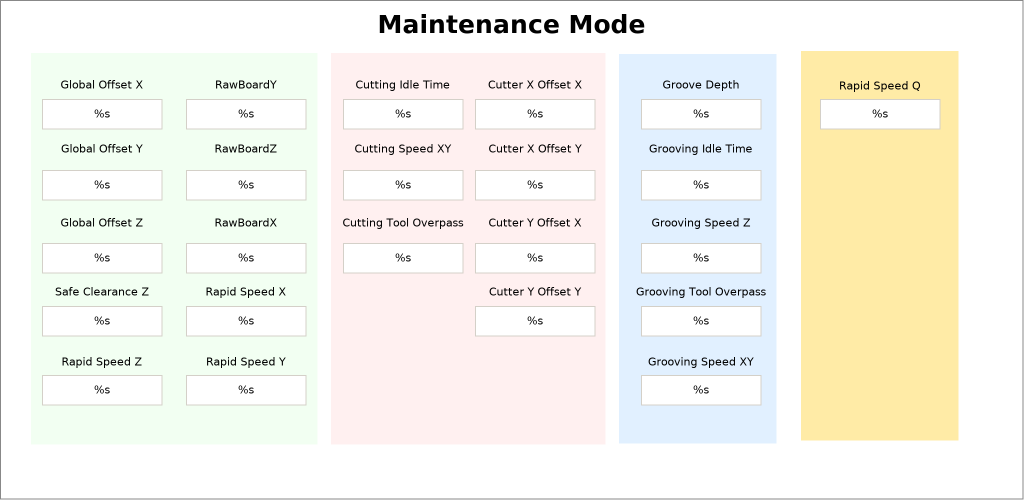
VISUALIZATION V_MaintenanceMode  // 1024x500
VAR_IN_OUT
	HMI : ST_PackMLBaseModule_HMI;
	HMI_GantryXYZ : ST_GantryXYZ_HMI;
	HMI_Recipe : ST_RecipeBuilder_HMI;
END_VAR
    Rectangle (30,52 288x393)
    Rectangle (330,52 276x393)
    Label (0,-1 1023x50), "Maintenance Mode"
    Rectangle (618,53 159x391)
    Textfield (641,99 120x30), "%s", text variable: HMI_Recipe.Config.GrooveDepthZ
        OnMouseClick: write the text variable via VisuDialogs.Numpad, min HMI_Recipe.Limits.GrooveDepthZ.MinVal, max HMI_Recipe.Limits.GrooveDepthZ.MaxVal
    Label (641,70 120x30), "Groove Depth"
    Textfield (641,306 120x30), "%s", text variable: HMI_Recipe.Config.GroovingOverpass
        OnMouseClick: write the text variable via VisuDialogs.Numpad, min HMI_Recipe.Limits.GroovingOverpass.MinVal, max HMI_Recipe.Limits.GroovingOverpass.MaxVal
    Label (641,277 120x30), "Grooving Tool Overpass"
    Textfield (641,375 120x30), "%s", text variable: HMI_GantryXYZ.Config.GroovingSpeedXY
        OnMouseClick: write the text variable via VisuDialogs.Numpad, min HMI_GantryXYZ.Limits.GroovingSpeedXY.MinVal, max HMI_GantryXYZ.Limits.GroovingSpeedXY.MaxVal
    Label (641,347 120x30), "Grooving Speed XY"
    Textfield (186,306 120x30), "%s", text variable: HMI_GantryXYZ.Config.RapidSpeedX
        OnMouseClick: write the text variable via VisuDialogs.Numpad, min HMI_GantryXYZ.Limits.RapidSpeedX.MinVal, max HMI_GantryXYZ.Limits.RapidSpeedX.MaxVal
    Label (186,277 120x30), "Rapid Speed X"
    Textfield (186,375 120x30), "%s", text variable: HMI_GantryXYZ.Config.RapidSpeedY
        OnMouseClick: write the text variable via VisuDialogs.Numpad, min HMI_GantryXYZ.Limits.RapidSpeedY.MinVal, max HMI_GantryXYZ.Limits.RapidSpeedY.MaxVal
    Label (186,347 120x30), "Rapid Speed Y"
    Textfield (641,243 120x30), "%s", text variable: HMI_GantryXYZ.Config.GroovingSpeedZ
        OnMouseClick: write the text variable via VisuDialogs.Numpad, min HMI_GantryXYZ.Limits.GroovingSpeedZ.MinVal, max HMI_GantryXYZ.Limits.GroovingSpeedZ.MaxVal
    Label (641,208 120x30), "Grooving Speed Z"
    Textfield (42,375 120x30), "%s", text variable: HMI_GantryXYZ.Config.RapidSpeedZ
        OnMouseClick: write the text variable via VisuDialogs.Numpad, min HMI_GantryXYZ.Limits.RapidSpeedZ.MinVal, max HMI_GantryXYZ.Limits.RapidSpeedZ.MaxVal
    Label (42,347 120x30), "Rapid Speed Z"
    Textfield (641,170 120x30), "%s", text variable: HMI_GantryXYZ.Config.GroovingIdleTime
        OnMouseClick: write the text variable via VisuDialogs.Numpad, min HMI_GantryXYZ.Limits.GroovingIdleTime.MinVal, max HMI_GantryXYZ.Limits.GroovingIdleTime.MaxVal
    Label (641,134 120x30), "Grooving Idle Time"
    Label (343,134 120x30), "Cutting Speed XY"
    Textfield (343,243 120x30), "%s", text variable: HMI_Recipe.Config.CuttingOverpass
        OnMouseClick: write the text variable via VisuDialogs.Numpad, min HMI_Recipe.Limits.CuttingOverpass.MinVal, max HMI_Recipe.Limits.CuttingOverpass.MaxVal
    Label (343,208 120x30), "Cutting Tool Overpass"
    Textfield (343,99 120x30), "%s", text variable: HMI_GantryXYZ.Config.CuttingIdleTime
        OnMouseClick: write the text variable via VisuDialogs.Numpad, min HMI_GantryXYZ.Limits.CuttingIdleTime.MinVal, max HMI_GantryXYZ.Limits.CuttingIdleTime.MaxVal
    Label (343,70 120x30), "Cutting Idle Time"
    Textfield (343,170 120x30), "%s", text variable: HMI_GantryXYZ.Config.CuttingSpeedXY
        OnMouseClick: write the text variable via VisuDialogs.Numpad, min HMI_GantryXYZ.Limits.CuttingSpeedXY.MinVal, max HMI_GantryXYZ.Limits.CuttingSpeedXY.MaxVal
    Label (475,70 120x30), "Cutter X Offset X"
    Textfield (475,170 120x30), "%s", text variable: HMI_GantryXYZ.Config.CutterXOffsetY
        OnMouseClick: write the text variable via VisuDialogs.Numpad, min HMI_GantryXYZ.Limits.CutterXOffsetY.MinVal, max HMI_GantryXYZ.Limits.CutterXOffsetY.MaxVal
    Label (475,134 120x30), "Cutter X Offset Y"
    Textfield (475,99 120x30), "%s", text variable: HMI_GantryXYZ.Config.CutterXOffsetX
        OnMouseClick: write the text variable via VisuDialogs.Numpad, min HMI_GantryXYZ.Limits.CutterXOffsetX.MinVal, max HMI_GantryXYZ.Limits.CutterXOffsetX.MaxVal
    Label (475,208 120x30), "Cutter Y Offset X"
    Textfield (475,306 120x30), "%s", text variable: HMI_GantryXYZ.Config.CutterYOffsetY
        OnMouseClick: write the text variable via VisuDialogs.Numpad, min HMI_GantryXYZ.Limits.CutterYOffsetY.MinVal, max HMI_GantryXYZ.Limits.CutterYOffsetY.MaxVal
    Label (475,277 120x30), "Cutter Y Offset Y"
    Textfield (475,243 120x30), "%s", text variable: HMI_GantryXYZ.Config.CutterYOffsetX
        OnMouseClick: write the text variable via VisuDialogs.Numpad, min HMI_GantryXYZ.Limits.CutterYOffsetX.MinVal, max HMI_GantryXYZ.Limits.CutterYOffsetX.MaxVal
    Label (42,70 120x30), "Global Offset X"
    Textfield (42,99 120x30), "%s", text variable: HMI_GantryXYZ.Config.GlobalOffsetX
        OnMouseClick: write the text variable via VisuDialogs.Numpad, min HMI_GantryXYZ.Limits.GlobalOffsetX.MinVal, max HMI_GantryXYZ.Limits.GlobalOffsetX.MaxVal
    Label (42,134 120x30), "Global Offset Y"
    Textfield (42,170 120x30), "%s", text variable: HMI_GantryXYZ.Config.GlobalOffsetY
        OnMouseClick: write the text variable via VisuDialogs.Numpad, min HMI_GantryXYZ.Limits.GlobalOffsetY.MinVal, max HMI_GantryXYZ.Limits.GlobalOffsetY.MaxVal
    Textfield (42,243 120x30), "%s", text variable: HMI_GantryXYZ.Config.GlobalOffsetZ
        OnMouseClick: write the text variable via VisuDialogs.Numpad, min HMI_GantryXYZ.Limits.GlobalOffsetZ.MinVal, max HMI_GantryXYZ.Limits.GlobalOffsetZ.MaxVal
    Label (42,208 120x30), "Global Offset Z"
    Textfield (186,243 120x30), "%s", text variable: HMI_GantryXYZ.Config.RawBoardX
        OnMouseClick: write the text variable via VisuDialogs.Numpad, min HMI_GantryXYZ.Limits.RawBoardX.MinVal, max HMI_GantryXYZ.Limits.RawBoardX.MaxVal
    Label (186,208 120x30), "RawBoardX"
    Textfield (186,99 120x30), "%s", text variable: HMI_GantryXYZ.Config.RawBoardY
        OnMouseClick: write the text variable via VisuDialogs.Numpad, min HMI_GantryXYZ.Limits.RawBoardY.MinVal, max HMI_GantryXYZ.Limits.RawBoardY.MaxVal
    Label (186,70 120x30), "RawBoardY"
    Textfield (186,170 120x30), "%s", text variable: HMI_GantryXYZ.Config.RawBoardZ
        OnMouseClick: write the text variable via VisuDialogs.Numpad, min HMI_GantryXYZ.Limits.RawBoardZ.MinVal, max HMI_GantryXYZ.Limits.RawBoardZ.MaxVal
    Label (186,134 120x30), "RawBoardZ"
    Textfield (42,306 120x30), "%s", text variable: HMI_GantryXYZ.Config.SafeClearanceZ
        OnMouseClick: write the text variable via VisuDialogs.Numpad, min HMI_GantryXYZ.Limits.SafeClearanceZ.MinVal, max HMI_GantryXYZ.Limits.SafeClearanceZ.MaxVal
    Label (42,277 120x30), "Safe Clearance Z"
    Rectangle (800,50 159x391)
    Textfield (820,99 120x30), "%s", text variable: HMI_GantryXYZ.Config.RapidSpeedQ
        OnMouseClick: write the text variable via VisuDialogs.Numpad, min HMI_GantryXYZ.Limits.RapidSpeedQ.MinVal, max HMI_GantryXYZ.Limits.RapidSpeedQ.MaxVal
    Label (820,71 120x30), "Rapid Speed Q"
END_VISUALIZATION

(* stored: Version 1.1.0.1, ProductVersion 3.1.4024.15
   Visu V_MaintenanceMode: Id {beddd7b9-7d38-4b95-a44e-95ac60c56cdb} *)
